VAR_GLOBAL
// Eingänge
net_licht_01 AT %I* : BOOL;
net_licht_02 AT %I* : BOOL;
net_licht_04 AT %I* : BOOL;
net_besucher_01 AT %I* : INT;
net_besucher_02 AT %I* : INT;
net_besucher_04 AT %I* : INT;
net_alarm_01 AT %I* : BOOL;
net_alarm_02 AT %I* : BOOL;
net_alarm_04 AT %I* : BOOL;
net_heizung_01 AT %I* : INT;
net_heizung_02 AT %I* : INT;
net_heizung_04 AT %I* : INT;


// Ausgänge
net_einbruch_alarm AT %Q* : BOOL;
net_reset_besucher AT %Q* : BOOL;
net_wind AT %Q* : REAL;
net_regen AT %Q* : REAL;
net_sonne AT %Q* : REAL;
net_heizung_out AT %Q* : INT;
END_VAR

(* stored: Version 1.1.0.1, ProductVersion 3.1.4018.5
   GVL Netzwerk: Id {e08085fc-300f-4b23-a231-42f824c44a9d} *)
